// TIA Portal V20 export
DATA_BLOCK "IDB_FB_ToggleDir"   // DB47
// stored: InstanceOfName ProductionLine.FB_ToggleDir, InstanceOfType FB, Namespace ProductionLine
"ProductionLine.FB_ToggleDir"
   // VAR
   //    "A1.12.1" { S7_SetPoint := 'True'} : "Global.ToggelDir";
   //    CurrentExpedtionDirection : Struct
   //       Straight : Bool;
   //       Left : Bool;
   //       None : Bool;
   //    END_STRUCT;
   //    CurrentStraightTableselection : Struct
   //       Table1 : Bool;
   //       Table2 : Bool;
   //       Table3 : Bool;
   //       Table4 : Bool;
   //       Table5 : Bool;
   //       None : Bool;
   //    END_STRUCT;
   //    CurrentLeftTableselection : Struct
   //       Table1 : Bool;
   //       Table2 : Bool;
   //       Table3 : Bool;
   //       Table4 : Bool;
   //       Table5 : Bool;
   //       None : Bool;
   //    END_STRUCT;
   // END_VAR
BEGIN
END_DATA_BLOCK
